INTERFACE IRecordDataQueue

METHOD write : BOOL
VAR_INPUT
	input_data	:T_Arg;
END_VAR
END_METHOD

END_INTERFACE

(* stored: Version 1.1.0.1, ProductVersion 3.1.4024.12
   Itf IRecordDataQueue: Id {31172c77-633a-46d5-b927-3b44dc9446a9}
   Method write: Id {b7310110-45a3-4bf4-930d-2690f31ed7d1} *)
